{attribute 'GeneratedUsingTerminal: EL2044-0000-0016'}
{attribute addProperty BoxType "EL2044-0000-0016"}
{attribute addProperty Id "OvertemperatureBOOL1Open_LoadBOOL1OvercurrentBOOL1Short_Circuit_to_24VBOOL1"}
{attribute addProperty CRC "3935122391"}
{attribute addProperty Size "4"}
TYPE Channel_EA8D33D7 :
STRUCT
	{attribute addProperty Name "Overtemperature"}
	Overtemperature : BOOL;
	{attribute addProperty Name "Open_Load"}
	Open_Load : BOOL;
	{attribute addProperty Name "Overcurrent"}
	Overcurrent : BOOL;
	{attribute addProperty Name "Short_Circuit_to_24V"}
	Short_Circuit_to_24V : BOOL;
END_STRUCT
END_TYPE

(* stored: Version 1.2.0.0, ProductVersion 3.1.4024.9
   DUT Channel_EA8D33D7: Id {dde087d0-6dc1-408a-84de-6d01c383d36a} *)
